PROGRAM MAIN
VAR
	bEnable : BOOL;
	bStart : BOOL;
END_VAR

bEnable:=bStart;
P_task1();

END_PROGRAM

(* stored: Version 1.1.0.1, ProductVersion 3.1.4024.12
   POU MAIN: Id {75da618d-82b5-4924-8926-19f065104ee3}, SpecialFunc None *)
